{attribute 'no_explicit_call' := 'do not call this function block directly'} 
FUNCTION_BLOCK CreateDirectory EXTENDS TOF_Core.Task
VAR
	{attribute 'OPC.UA.DA' := '0'}
	_ClassName : STRING := __POUNAME();

	{attribute 'OPC.UA.DA' := '0'}
    _CreateDirectory : Tc2_System.FB_CreateDir;
END_VAR

{attribute 'monitoring' := 'call'}
{attribute 'OPC.UA.DA.Property' := '1'}
{attribute 'OPC.UA.DA' := '1'}
PROPERTY AmsNetId : Tc2_System.T_AmsNetID
GET
AmsNetId := _CreateDirectory.sNetId;
END_GET
SET
_CreateDirectory.sNetId := AmsNetId;
END_SET
END_PROPERTY

{attribute 'monitoring' := 'call'}
PROPERTY ClassName : STRING
GET
ClassName := _ClassName;
END_GET
END_PROPERTY

{attribute 'monitoring' := 'call'}
{attribute 'OPC.UA.DA.Property' := '1'}
{attribute 'OPC.UA.DA' := '1'}
PROPERTY DirectoryPath : Tc2_System.T_MaxString
GET
DirectoryPath := _CreateDirectory.sPathName;
END_GET
SET
_CreateDirectory.sPathName := DirectoryPath;
END_SET
END_PROPERTY

{attribute 'monitoring' := 'call'}
PROPERTY NamespaceName : STRING
GET
NamespaceName := CurrentNamespace.Name;
END_GET
END_PROPERTY

METHOD PROTECTED OnCancel
_CreateDirectory(bExecute := FALSE);
END_METHOD

METHOD PROTECTED OnRunning 
VAR_INPUT
	startRequest : BOOL;
END_VAR
VAR_OUTPUT
	state : TASK_RUNNING_STATE;
END_VAR
VAR
	propertyNotSpecifiedException :	DataMemberNotSpecifiedException;
	createDirectoryException : TOF_Core.StandardException;
	errorMessageBuilder : TOF_Core.WideStringBuilder;
END_VAR
IF startRequest THEN 
	IF TOF_Core.StringHelper.IsNullOrWhiteSpace(_CreateDirectory.sPathName) THEN
		propertyNotSpecifiedException.Throw(NamespaceName, ClassName, __POUNAME(), __POSITION(), 'DirectoryPath');		
	END_IF
	
	_CreateDirectory(bExecute := FALSE);
END_IF

_CreateDirectory(bExecute := TRUE);

IF _CreateDirectory.bError THEN
	errorMessageBuilder
		.AppendString("An error occurred while creating the directory '")
		.Append(_CreateDirectory.sPathName)
		.AppendString("'");

	createDirectoryException.Throw(NamespaceName, ClassName, __POUNAME(), __POSITION(), errorMessageBuilder.ToString());
END_IF

IF NOT _CreateDirectory.bBusy THEN
	state := TOF_Core.TASK_RUNNING_STATE.DONE;
END_IF
END_METHOD

{attribute 'monitoring' := 'call'}
{attribute 'OPC.UA.DA.Property' := '1'}
{attribute 'OPC.UA.DA' := '1'}
PROPERTY PathType : Tc2_System.E_OpenPath
GET
PathType := _CreateDirectory.ePath;
END_GET
SET
_CreateDirectory.ePath := PathType;
END_SET
END_PROPERTY

{attribute 'monitoring' := 'call'}
PROPERTY Size : ULINT
GET
Size := XSIZEOF(THIS^);
END_GET
END_PROPERTY

{attribute 'monitoring' := 'call'}
{attribute 'OPC.UA.DA.Property' := '1'}
{attribute 'OPC.UA.DA' := '1'}
PROPERTY Timeout : TIME
GET
Timeout := _CreateDirectory.tTimeout;
END_GET
SET
_CreateDirectory.tTimeout := Timeout;
END_SET
END_PROPERTY

END_FUNCTION_BLOCK

(* stored: Version 1.1.0.1
   POU CreateDirectory: Id {7b0b8920-cd1b-44d1-9ca2-1004e427656c}, SpecialFunc None
   Folder Members to override: Id {740079d8-792c-4051-b807-b10023f9c7a1}
   Property AmsNetId: Id {ed338df4-10dc-451a-b64d-a000a295e7f0}
   Get Get: Id {94b5c541-fb9b-4788-a387-16d6d7a06a3f}
   Set Set: Id {477e135b-e114-4f7b-ae5e-413843dd690f}
   Property ClassName: Id {68947efb-286a-42af-a556-a0bbd5d3027a}
   Get Get: Id {40a07058-94c4-4be0-ab88-a373f33d3011}
   Property DirectoryPath: Id {7d34ff6b-66c9-43e2-9ce1-01d401372e05}
   Get Get: Id {bfb35ddc-0143-4123-989c-469790325d20}
   Set Set: Id {f1f98b86-e1b0-48a8-a264-70f11718c110}
   Property NamespaceName: Id {ea279b18-2495-419a-af6e-f1db1538b308}
   Get Get: Id {affba913-0ba6-4588-83ed-6a9649f3e1dc}
   Method OnCancel: Id {914b9647-4a97-4ca9-943b-d06999c3b774}
   Method OnRunning: Id {6bd810fa-872b-4e47-b2bc-32ff3c16f403}
   Property PathType: Id {813cddba-24ae-417e-a32e-8078530fc9b5}
   Get Get: Id {26543d70-59ee-403c-af69-d4faa3e2e712}
   Set Set: Id {fc38db83-a1b0-4341-9146-45fe2533fa6e}
   Property Size: Id {ff29508a-b927-484d-8776-c7a1fd61b57a}
   Get Get: Id {9fd144e1-4541-4668-9bfe-274b7a79cf1d}
   Property Timeout: Id {78fb4594-c887-4181-a8a6-4363e1f0945e}
   Get Get: Id {8affc407-c0f2-46cc-acef-d2a177ecaf4b}
   Set Set: Id {0f89e125-a68f-47d7-ab94-803cd70c6f9c} *)
